// TIA Portal V18 export
DATA_BLOCK "gDb_LED_state"   // DB9
{ S7_Optimized_Access := 'TRUE' }
VERSION : 0.1
// stored: AutoNumber true, DBAccessibleFromOPCUA true, DBAccessibleFromWebserver true, IsOnlyStoredInLoadMemory false, IsRetainMemResEnabled false, IsWriteProtectedInAS false, MemoryReserve 100
   VAR RETAIN
      green : Bool;
      yellow : Bool;
      red : Bool;
   END_VAR
BEGIN
END_DATA_BLOCK
